// TIA Portal V19 export
DATA_BLOCK "Rollformer"   // DB141
// stored: InstanceOfName Rollformer_FB, InstanceOfType FB
"Rollformer_FB"
   // VAR_INPUT
   //    AreaInterface : "AreaInterface";
   //    ZSI : "udt_ZoneSafetyInterface";
   //    DSI : "udt_DeviceSafetyInterface";
   //    Drive : "TAx_DriveInterface";
   //    DataIn : Struct
   //       Feed : "PositioningMachine_DataIn";
   //       ConnectorPlugged1 : Bool;
   //       ConnectorPlugged2 : Bool;
   //       ConnectorPlugged3Side1 : Bool;
   //       ConnectorPlugged3Side2 : Bool;
   //    END_STRUCT;
   //    CIn : Struct
   //       ExtEnable_LoopFwdOk : Bool;
   //       ExtEnable_LoopBwdOk : Bool;
   //       ExtEnable_FlyingShareOk : Bool;
   //       ExtEnable_MaterialCounterOK : Bool;
   //       ExtEnable_UnloadRollwayOk : Bool;
   //       ExtEnable_MwFakCalcOk : Bool;
   //       Loop1_VelOverride : LReal;
   //       SOS_Enable : Bool;
   //       Manager : "PositioningMachine_Manager";
   //    END_STRUCT;
   //    Config : Struct
   //       Feed : "PositioningMachine_Config";
   //       Data : "PositioningMachine_Ax_Parameters";
   //       DataPresence : Bool;
   //    END_STRUCT;
   // END_VAR
   // VAR_OUTPUT
   //    MachineInterface : "MachineInterface";
   //    COut : Struct
   //       Feed : "PositioningMachine_COut";
   //       EnableSOS : Bool;
   //    END_STRUCT;
   //    DataOut : Struct
   //       Feed : "PositioningMachine_DataOut";
   //    END_STRUCT;
   // END_VAR
   // VAR_IN_OUT
   //    TO_Ax : TO_PositioningAxis;
   //    PersistentValues : "udt_Rollformer_Pers";
   // END_VAR
   // VAR
   //    Alarms : Struct
   //       Feed : "PositioningMachine_Alr";
   //       ConnectorNotPlugged1 : Bool;
   //       ConnectorNotPlugged2 : Bool;
   //       ConnectorNotPlugged3Side1 : Bool;
   //       ConnectorNotPlugged3Side2 : Bool;
   //    END_STRUCT;
   //    Warnings : Struct
   //       Feed : "PositioningMachine_Wng";
   //       ExtraLowIsON : Bool;
   //       MissingCnd : Struct
   //          FlyingShare : Bool;
   //          MaterialCounter : Bool;
   //          UnloadRollway : Bool;
   //          MwFakClac : Bool;
   //          Loop1_Enable_BWD : Bool;
   //          Loop1_Enable_FWD : Bool;
   //       END_STRUCT;
   //    END_STRUCT;
   //    HMI : Struct
   //       MissingCnd : Struct
   //          FlyingShare : Bool;
   //          MaterialCounter : Bool;
   //          UnloadRollway : Bool;
   //          MwFacCalc : Bool;
   //          Loop1_Enable_BWD : Bool;
   //          Loop1_Enable_FWD : Bool;
   //       END_STRUCT;
   //       ManTargetMaterialPosition : LReal;
   //    END_STRUCT;
   //    Sts : Struct
   //       CndBWD_OK : Bool;
   //       CndFWD_OK : Bool;
   //    END_STRUCT;
   //    Feed : "PositioningMachine_FB";
   //    TON_SOS : TON_TIME;
   // END_VAR
BEGIN
END_DATA_BLOCK
